PROGRAM P01_BottleSorter
VAR
END_VAR

aBottleSorterWarnings();

ACTION aBottleSorterWarnings:
//Warning 0

IF (stBottleSorterRead.eReservedSignals.iReserved20.0 AND stBottleSorterRead.bEnable) AND NOT BottleSorterWarning[0].bWarning THEN
	BottleSorterWarning[0].bWarning											:=TRUE;
	BottleSorterWarning[0].udiWarningCode									:=9;
	BottleSorterWarning[0].sDescription										:='Sorter butelek | Brak butelek w zasobniku';
ELSIF NOT stBottleSorterRead.eReservedSignals.iReserved20.0 AND BottleSorterWarning[0].bAcknowledge THEN
	BottleSorterWarning[0].bWarning											:=FALSE;
	BottleSorterWarning[0].bAcknowledge										:=FALSE;
	VIS.uliWarningAcknowledge.33											:=FALSE;
ELSIF BottleSorterWarning[0].bAcknowledge THEN                                
	BottleSorterWarning[0].bAcknowledge										:=TRUE;
END_IF

//Warning 1
IF stBottleSorterRead.eReservedSignals.iReserved20.1 AND NOT BottleSorterWarning[1].bWarning THEN
	BottleSorterWarning[1].bWarning											:=TRUE;
	BottleSorterWarning[1].udiWarningCode									:=10;
	BottleSorterWarning[1].sDescription										:='Sorter butelek | warning 1';
ELSIF NOT stBottleSorterRead.eReservedSignals.iReserved20.1 AND BottleSorterWarning[1].bAcknowledge THEN
	BottleSorterWarning[1].bWarning											:=FALSE;
	BottleSorterWarning[1].bAcknowledge										:=FALSE;
	VIS.uliWarningAcknowledge.34											:=FALSE;
ELSIF BottleSorterWarning[1].bAcknowledge THEN                                
	BottleSorterWarning[1].bAcknowledge										:=TRUE;
END_IF

//Warning 2
IF stBottleSorterRead.eReservedSignals.iReserved20.2 AND NOT BottleSorterWarning[2].bWarning THEN
	BottleSorterWarning[2].bWarning											:=TRUE;
	BottleSorterWarning[2].udiWarningCode									:=11;
	BottleSorterWarning[2].sDescription										:='Sorter butelek | warning 2';
ELSIF NOT stBottleSorterRead.eReservedSignals.iReserved20.1 AND BottleSorterWarning[2].bAcknowledge THEN
	BottleSorterWarning[2].bWarning											:=FALSE;
	BottleSorterWarning[2].bAcknowledge										:=FALSE;
	VIS.uliWarningAcknowledge.35											:=FALSE;
ELSIF BottleSorterWarning[2].bAcknowledge THEN                                
	BottleSorterWarning[2].bAcknowledge										:=TRUE;
END_IF

//Warning 3
IF stBottleSorterRead.eReservedSignals.iReserved20.3 AND NOT BottleSorterWarning[3].bWarning THEN
	BottleSorterWarning[3].bWarning											:=TRUE;
	BottleSorterWarning[3].udiWarningCode									:=12;
	BottleSorterWarning[3].sDescription										:='Sorter butelek | warning 3';
ELSIF NOT stBottleSorterRead.eReservedSignals.iReserved20.1 AND BottleSorterWarning[3].bAcknowledge THEN
	BottleSorterWarning[3].bWarning											:=FALSE;
	BottleSorterWarning[3].bAcknowledge										:=FALSE;
	VIS.uliWarningAcknowledge.36											:=FALSE;
ELSIF BottleSorterWarning[3].bAcknowledge THEN                                
	BottleSorterWarning[3].bAcknowledge										:=TRUE;
END_IF

//Warning 4
IF stBottleSorterRead.eReservedSignals.iReserved20.4 AND NOT BottleSorterWarning[4].bWarning THEN
	BottleSorterWarning[4].bWarning											:=TRUE;
	BottleSorterWarning[4].udiWarningCode									:=13;
	BottleSorterWarning[4].sDescription										:='Sorter butelek | warning 4';
ELSIF NOT stBottleSorterRead.eReservedSignals.iReserved20.1 AND BottleSorterWarning[4].bAcknowledge THEN
	BottleSorterWarning[4].bWarning											:=FALSE;
	BottleSorterWarning[4].bAcknowledge										:=FALSE;
	VIS.uliWarningAcknowledge.37											:=FALSE;
ELSIF BottleSorterWarning[4].bAcknowledge THEN
	BottleSorterWarning[4].bAcknowledge										:=TRUE;
END_IF

//Warning 5
IF stBottleSorterRead.eReservedSignals.iReserved20.5 AND NOT BottleSorterWarning[5].bWarning THEN
	BottleSorterWarning[5].bWarning											:=TRUE;
	BottleSorterWarning[5].udiWarningCode									:=14;
	BottleSorterWarning[5].sDescription										:='Sorter butelek | warning 5';
ELSIF NOT stBottleSorterRead.eReservedSignals.iReserved20.1 AND BottleSorterWarning[5].bAcknowledge THEN
	BottleSorterWarning[5].bWarning											:=FALSE;
	BottleSorterWarning[5].bAcknowledge										:=FALSE;
	VIS.uliWarningAcknowledge.38											:=FALSE;
ELSIF BottleSorterWarning[5].bAcknowledge THEN
	BottleSorterWarning[5].bAcknowledge										:=TRUE;
END_IF
END_ACTION

END_PROGRAM

(* stored: Version 1.1.0.1, ProductVersion 3.1.4026.13, FileIdentifier 10ad54e3022875e8cc3cc7eda35dae2ddf4115e8, FileSignature 0dc5d2d959a61fa12bed3cdf5cf95dbf53b97f50b9724c4e2ca6ad0baf63d7788c5de88e2a7b69be93cf02b888f9e809754e6e3750f641cfae9c82feca6496c6d0ef2e4c6a2a776aa854502e2fec50907d6b9d8b6d1ce53577904883f085a3470f3fafb1e5269e79f35d417d8281b66f42b4996183b519b3d5ea93090661f4dd02a41a9ba8debeda5f1cfc3b8761aee71d02a179f3231dd3d058aba9e67cc4497b802a123ee2a1ef402844b0d5b9eaf771a8bad2bf7d0d5093f1e487f6cc9638bfae6bd8a0003c05c12aff05501c16892366cea5474371b26715190b6d362fabefdbcd80a7016dc6bb233de8160d7bfafdd4d9e255b6d8355537f5bc4d23a6a4
   POU P01_BottleSorter: Id {0c65c720-242f-464e-b6dd-b5c8a3ae5224}, SpecialFunc None
   Action aBottleSorterWarnings: Id {eeea2c8b-73bf-4166-9f2e-9ca266f1b865} *)
